// Annex I I.3/I.5 - the Staubli VAL3 connector over the SIM channel. No socket,
// no emulator, no arm: FB_SimByteChannel scripts request/reply pairs, so the wire
// protocol and every refusal path are provable in CI (S5.7, Annex H).
//
// This is the transport-layer half of the I.5c simulation requirement. The SRS
// Emulator remains the higher-fidelity layer for motion behaviour; what is proven
// here is the part that must hold before an emulator is worth starting: that the
// connector speaks the agreed frames, and that it REFUSES rather than pretends
// when the link is down, the mode is wrong, or the path was left.
//
// Linked means session up AND heartbeat healthy (Core §3.15.2), and the heartbeat
// is the TON-driven status poll, so every test that needs a live link runs ACROSS
// SCANS and scripts the STA reply the heartbeat asks for.
FUNCTION_BLOCK FB_RobotConnector_Tests EXTENDS TcUnit.FB_TestSuite
VAR
    _chan  : FB_SimByteChannel;
    _conn  : FB_StaubliVal3Connector;
    _chanB : FB_SimByteChannel;
    _connB : FB_StaubliVal3Connector;
    _chanC : FB_SimByteChannel;
    _connC : FB_StaubliVal3Connector;
    _chanD : FB_SimByteChannel;
    _connD : FB_StaubliVal3Connector;
    _ok    : BOOL;
    _i, _i2, _i4 : INT;
    _diag  : ST_Diagnostic;   // C0185: cannot access .member on a property result
    _pose  : ST_RobotPose;
    _w1, _w2, _w3, _w4, _w5, _w6 : BOOL;
    _sent2, _sent4 : BOOL;
END_VAR

Link_down_refuses_every_command_rather_than_dropping_it();
Id_addressed_commands_are_framed_on_the_wire();
Status_poll_publishes_the_controllers_reported_facts();
Controller_error_is_carried_verbatim_and_faults();
Resume_is_refused_when_the_arm_left_the_retained_path();
Unknown_mode_request_is_refused_outright();

METHOD PRIVATE Link_down_refuses_every_command_rather_than_dropping_it
TEST('Link_down_refuses_every_command_rather_than_dropping_it');
IF NOT _w1 THEN
    // Deliberately never set up or connected: there is no session.
    // A command issued now must come back FALSE. Silently queueing it would let a
    // sequence wait on a robot that never heard the command (Annex D).
    AssertFalse(Condition := _connB.PowerOn(),
        Message := 'a command on a down link is refused, not queued');
    AssertFalse(Condition := _connB.MoveToPoint(PointId := 7),
        Message := 'and so is an ID-addressed move');
    AssertFalse(Condition := _connB.Linked,
        Message := 'Linked reports the link honestly');
    _diag := _connB.LastResult;
    AssertEquals_DINT(Expected := E_Reason.LINK_TIMEOUT, Actual := _diag.ReasonCode,
        Message := 'the refusal carries the link reason for the CM to adopt');
    _w1 := TRUE;
END_IF
TEST_FINISHED();
END_METHOD

METHOD PRIVATE Id_addressed_commands_are_framed_on_the_wire
TEST('Id_addressed_commands_are_framed_on_the_wire');
IF _w2 THEN
    TEST_FINISHED();
    RETURN;
END_IF
IF _i2 = 0 THEN
    // The channel only replies when the sent line matches EXACTLY, so a reply
    // proves the frame. Every argument is an identifier - never a coordinate (I.1).
    _chan.Script(Expect := 'STA$R', Reply := 'STA,OK,0,1,AUTO,4,0,1,0,0,0,0,0,0$R');
    _chan.Script(Expect := 'TPL,11,22$R', Reply := 'TPL,OK$R');
    _conn.SetupLink(Name := 'Test.Robot', Chan := _chan, DevHost := '10.0.0.20', DevPort := 11000);
    _conn.Connect();
END_IF
_conn.Cyclic();
_i2 := _i2 + 1;
IF _conn.Linked AND NOT _sent2 THEN
    AssertTrue(Condition := _conn.MoveTemplate(FromPosId := 11, ToPosId := 22),
        Message := 'a routed move is accepted and framed as TPL,from,to');
    _sent2 := TRUE;
ELSIF _sent2 AND (_conn.LastResponse = 'TPL,OK') THEN
    AssertEquals_STRING(Expected := 'TPL,OK', Actual := _conn.LastResponse,
        Message := 'and the controller acknowledgement is published');
    _w2 := TRUE;
    TEST_FINISHED();
ELSIF _i2 > 1000 THEN
    AssertTrue(Condition := FALSE,
        Message := 'the link never came up, or the framed move was never acknowledged');
    _w2 := TRUE;
    TEST_FINISHED();
END_IF
END_METHOD

METHOD PRIVATE Status_poll_publishes_the_controllers_reported_facts
TEST('Status_poll_publishes_the_controllers_reported_facts');
// The poll is the TON-driven heartbeat, so this test must run ACROSS SCANS - a loop
// of Cyclic() calls inside one scan advances no time and the timer never fires.
// Same shape as FB_TcpDev_Tests.Timeout_faults_10402, for the same reason.
IF _w3 THEN
    TEST_FINISHED();
    RETURN;
END_IF
IF _i = 0 THEN
    // STA,OK,busy,ref,mode,area,prot,resumable,x,y,z,rx,ry,rz
    _chanC.Script(Expect := 'STA$R',
        Reply := 'STA,OK,0,1,AUTO,4,0,1,100.5,200,300,0,0,90$R');
    _connC.SetupLink(Name := 'Test.RobotC', Chan := _chanC, DevHost := '10.0.0.21', DevPort := 11000);
    _connC.Connect();
END_IF
_connC.Cyclic();
_i := _i + 1;

IF _connC.Referenced THEN
    // Referenced only becomes TRUE once a status reply was parsed, so reaching
    // here proves the heartbeat fired, framed STA, and the reply was decoded.
    AssertTrue(Condition := _connC.Linked,
        Message := 'an answered status poll is a healthy heartbeat: the link is up');
    AssertTrue(Condition := _connC.ActualMode = E_RobotOpMode.AUTO_REMOTE,
        Message := 'ActualMode is what the controller REPORTS, not what we asked for');
    AssertEquals_DWORD(Expected := 4, Actual := _connC.CurrentArea,
        Message := 'the planning area is published for area-resolved motion');
    AssertFalse(Condition := _connC.ProtectiveStop,
        Message := 'the protective stop is published separately from S9 safety');
    _pose := _connC.ActualPosition;
    AssertEquals_LREAL(Expected := 100.5, Actual := _pose.X, Delta := 0.001,
        Message := 'the live pose is readable for display and diagnostics');
    AssertEquals_LREAL(Expected := 90, Actual := _pose.RZ, Delta := 0.001,
        Message := 'including orientation');
    // Jogging is bounded by the CONTROLLER's mode, not by a PLC release alone.
    // Asserted here because this is where a LINKED connector reporting AUTO
    // exists - proving the refusal comes from the mode gate and not the link.
    AssertFalse(Condition := _connC.Jog(Mode := E_RobotJogMode.JOINT, Axis := 1, Dir := 1),
        Message := 'jogging is refused while the controller reports auto');
    _w3 := TRUE;
    TEST_FINISHED();
ELSIF _i > 1000 THEN
    // Bounded so a regression fails loudly here instead of hanging the runner
    // with no message, which is the worse failure.
    AssertTrue(Condition := FALSE,
        Message := 'the status poll never delivered a reply');
    _w3 := TRUE;
    TEST_FINISHED();
END_IF
END_METHOD

METHOD PRIVATE Controller_error_is_carried_verbatim_and_faults
TEST('Controller_error_is_carried_verbatim_and_faults');
IF _w4 THEN
    TEST_FINISHED();
    RETURN;
END_IF
IF _i4 = 0 THEN
    _chanD.Script(Expect := 'STA$R', Reply := 'STA,OK,0,0,AUTO,0,0,0,0,0,0,0,0,0$R');
    _chanD.Script(Expect := 'HOME$R', Reply := 'HOME,ERR,J12,joint 3 out of range$R');
    _connD.SetupLink(Name := 'Test.RobotD', Chan := _chanD, DevHost := '10.0.0.22', DevPort := 11000);
    _connD.Connect();
END_IF
_connD.Cyclic();
_i4 := _i4 + 1;
_diag := _connD.ControllerMessage;
IF _connD.Linked AND NOT _sent4 THEN
    AssertTrue(Condition := _connD.Home(), Message := 'the request is accepted by the transport');
    _sent4 := TRUE;
ELSIF _sent4 AND (_diag.ReasonCode = PL_ModuleReasons.ROBOT_CONTROLLER_FAULT) THEN
    // The robot's OWN text survives. Paraphrasing it would cost the technician the
    // one string that identifies the fault on the pendant (S8.2).
    AssertTrue(Condition := FIND(_diag.Description, 'joint 3 out of range') > 0,
        Message := 'the controller message is carried verbatim');
    _diag := _connD.LastResult;
    AssertEquals_DINT(Expected := PL_ModuleReasons.ROBOT_CONTROLLER_FAULT,
        Actual := _diag.ReasonCode,
        Message := 'and it is the refusal the robot CM adopts as its first-out');
    AssertFalse(Condition := _connD.MotionBusy,
        Message := 'a refused command does not leave the connector claiming motion');
    _w4 := TRUE;
    TEST_FINISHED();
ELSIF _i4 > 1000 THEN
    AssertTrue(Condition := FALSE,
        Message := 'the controller error never arrived');
    _w4 := TRUE;
    TEST_FINISHED();
END_IF
END_METHOD

METHOD PRIVATE Resume_is_refused_when_the_arm_left_the_retained_path
TEST('Resume_is_refused_when_the_arm_left_the_retained_path');
IF NOT _w5 THEN
    // Resumable=0 in the status reply. A hold is exactly when an operator jogs the
    // arm, and resuming onto a path the tool has left is how a robot drives through
    // a fixture - so this must refuse rather than execute (I.4b).
    AssertFalse(Condition := _connD.Resumable,
        Message := 'the connector reports resumption invalid by default');
    AssertFalse(Condition := _connD.Resume(),
        Message := 'and Resume is refused rather than sent');
    _w5 := TRUE;
END_IF
TEST_FINISHED();
END_METHOD

METHOD PRIVATE Unknown_mode_request_is_refused_outright
TEST('Unknown_mode_request_is_refused_outright');
IF NOT _w6 THEN
    // Requesting UNKNOWN is meaningless and must never reach the controller: an
    // uninitialised or unparsed mode must not travel as though it were a real
    // request. Self-contained on purpose - the previous version asserted a
    // precondition owned by another test, so one root cause failed two tests.
    AssertFalse(Condition := _connB.RequestMode(Mode := E_RobotOpMode.UNKNOWN),
        Message := 'an UNKNOWN mode request is refused before the transport');
    _w6 := TRUE;
END_IF
TEST_FINISHED();
END_METHOD

END_FUNCTION_BLOCK

(* stored: Version 1.1.0.1, ProductVersion 3.1.4024.12
   POU FB_RobotConnector_Tests: Id {dc5e0fca-eaee-44bb-a584-b0c619ee9c62}, SpecialFunc None
   Method Link_down_refuses_every_command_rather_than_dropping_it: Id {ce24fe50-b1bd-4599-ac24-7c1223c8a3f1}
   Method Id_addressed_commands_are_framed_on_the_wire: Id {7d6065f0-81a1-434b-a53e-2d75346f7635}
   Method Status_poll_publishes_the_controllers_reported_facts: Id {fa78ee37-e9e9-4f21-b601-5281d6c921be}
   Method Controller_error_is_carried_verbatim_and_faults: Id {6b3683ef-43c0-4588-8bb8-8cc304187f2f}
   Method Resume_is_refused_when_the_arm_left_the_retained_path: Id {b4d21257-73b9-41d0-b9fd-e98a9902a534}
   Method Unknown_mode_request_is_refused_outright: Id {1558bc16-a131-4003-9497-4383dd2e5e51} *)
